PROGRAM MAIN
VAR
	fbMotion1: fbMotion;
	fbMotion2: fbMotion;

	sAxis1	:	ST_Axis;
	sAxis2	:	ST_Axis;
		
	fbCAM_IN: MC_CamIn;
	fbCAM_OUT: MC_CamOut;
	

	bCamIN	:	BOOL;
	bCamOutDone	:	BOOL;
	
	nCamTableID	:	UDINT	:=	1;
	bCamSync: BOOL;
	scaling	:	ST_CamScalingData;
	
	nstate: INT;
	bExe: BOOL;
END_VAR


fbMotion1(stAxis:=sAxis1 , axis:=axis1 );
fbMotion2(stAxis:=sAxis2 , axis:= axis2);

ACT_Motion();
ACT_CAM();

ACTION ACT_CAM:
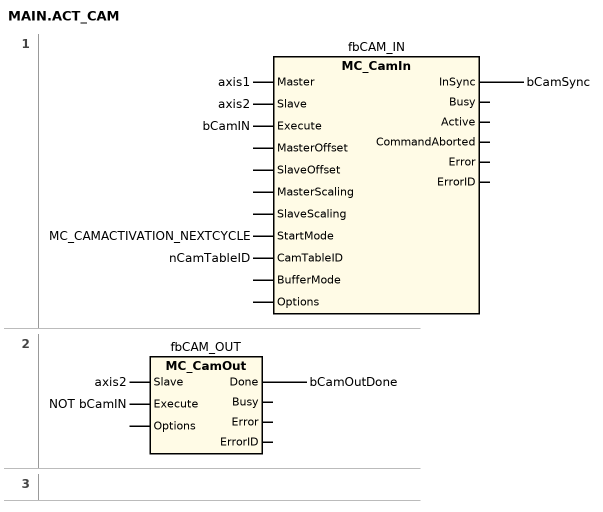
// NETWORK 1
fbCAM_IN(
    Master := axis1,
    Slave := axis2,
    Execute := bCamIN,
    StartMode := MC_CAMACTIVATION_NEXTCYCLE,
    CamTableID := nCamTableID); // MC_CamIn
bCamSync := fbCAM_IN.InSync;

// NETWORK 2
fbCAM_OUT(Slave := axis2, Execute := NOT bCamIN); // MC_CamOut
bCamOutDone := fbCAM_OUT.Done;

// NETWORK 3
END_ACTION

ACTION ACT_Motion:

saxis1.INPUT.nOverride	:=	100;
saxis2.INPUT.nOverride	:=	100;

CASE nstate	OF
	
	0:
	
		IF bExe	THEN
			nState	:=1;
			
			saxis1.INPUT.bPowerEnable	:=TRUE;
			saxis2.INPUT.bPowerEnable	:=TRUE;
		
			saxis1.INPUT.bStopEnable	:=	FALSE;
			saxis2.INPUT.bStopEnable	:=	FALSE;
			
			saxis1.INPUT.bMoveAbs	:=	FALSE;

			bCamIN	:=	FALSE;

		END_IF
		
	1:
		IF saxis1.OUTPUT.bPowerStat THEN
			nState	:=	10;
		END_IF	
		
	10:
		saxis1.INput.fPosition	:=	0;
		saxis1.INPUT.fVelo	:=	4000;
		saxis1.INPUT.bMoveAbs	:=	TRUE;
		
		saxis1.INPUT.bStopEnable	:=	FALSE;
		saxis2.INPUT.bStopEnable	:=	FALSE;
		
			IF	saxis1.OUTPUT.bMoveAbsBusy 
			AND NOT saxis1.OUTPUT.bMoveAbsErr	THEN
				
				nState	:=	20;
				
			ELSIF	saxis1.OUTPUT.bMoveAbsErr
			OR	saxis2.OUTPUT.bMoveAbsErr THEN
			
				nState	:=	999;
				
			END_IF
			
	20:
			IF saxis1.OUTPUT.bMoveAbsDone
			AND NOT saxis1.OUTPUT.bMoveAbsErr	THEN
				
				saxis1.INPUT.bMoveAbs	:=	FALSE;
				nState	:=	21;
								
			ELSIF	saxis1.OUTPUT.bMoveAbsErr
			OR	saxis2.OUTPUT.bMoveAbsErr THEN
				nState	:=	999;
			END_IF
			
	21:
		IF	saxis2.OUTPUT.bPowerStat	THEN
			nState	:=	22;
		END_IF
		
	22:
		bCamIN	:=	TRUE;
		IF bCamSync THEN
			nstate:=30;
		END_IF
	
	30:
		saxis1.INPUT.fPosition	:=	1800;
		saxis1.INPUT.fVelo	:=	1200;
		saxis1.INPUT.bMoveAbs	:=	TRUE;
		saxis1.INPUT.bStopEnable	:=	FALSE;
		saxis2.INPUT.bStopEnable	:=	FALSE;
		
			
			IF	(saxis1.OUTPUT.bMoveAbsBusy 
			AND NOT saxis1.OUTPUT.bMoveAbsErr 
			AND NOT	saxis1.OUTPUT.bPowerError)	THEN
				nState	:=	40;
			ELSIF	saxis1.OUTPUT.bMoveAbsErr
			OR	saxis2.OUTPUT.bMoveAbsErr THEN
				nState	:=	999;
			END_IF
			
	40:
			IF saxis1.OUTPUT.bMoveAbsDone
			AND NOT saxis1.OUTPUT.bMoveAbsErr 
			AND NOT	saxis1.OUTPUT.bPowerError	THEN
				
				saxis1.INPUT.bMoveAbs	:=	FALSE;
				nState	:=	0;
								
			ELSIF	saxis1.OUTPUT.bMoveAbsErr
			OR	saxis2.OUTPUT.bMoveAbsErr THEN
				nState	:=	999;
			END_IF
		
END_CASE

IF NOT bExe THEN
	
				saxis1.INPUT.bMoveAbs	:=	FALSE;
				saxis1.INPUT.bStopEnable	:=	TRUE;
				saxis2.INPUT.bStopEnable	:=	TRUE;
				
				IF saxis1.OUTPUT.bStopDone	AND	saxis2.OUTPUT.bStopDone THEN
				nState	:=	0;
				END_IF
END_IF

IF saxis1.OUTPUT.bPowerError	OR	saxis2.OUTPUT.bPowerError	THEN
	
	saxis1.INPUT.bReset	:=	TRUE;
	saxis2.INPUT.bReset	:=	TRUE;

	saxis1.INPUT.bMoveAbs	:=	FALSE;
	saxis2.INPUT.bMoveAbs	:=	FALSE;

	IF saxis1.OUTPUT.bResetDone	AND	saxis2.OUTPUT.bResetDone	THEN
	nState	:=	0;
	END_IF	
END_IF
END_ACTION

END_PROGRAM

(* stored: Version 1.1.0.1, ProductVersion 3.1.4022.18
   POU MAIN: Id {4aed3cb2-ff68-4837-9efa-f60baf4bb5af}, SpecialFunc None
   Action ACT_CAM: Id {ac6841b7-425c-4c21-8d3a-97a2aa6c1e09}
   Action ACT_Motion: Id {cb5c0343-74f6-427b-8ad4-046ad1eb71ea} *)
